// TIA Portal project "2Nastri1Ruota" (V17)
// Vorlageprojekt für das Buch mit Zielsystem S7-1200

(* hardware
DEVICE "S7-1200-Station_1"  S7-1200 Station
   slot 0: "Baugruppenträger_0"  Rack  V1.0
   slot 1: "PLC_1"  CPU 1211C DC/DC/DC  6ES7 211-1AE40-0XB0  V4.1
*)

// ===== PLC "PLC_1"  CPU 1211C DC/DC/DC =====

VAR_GLOBAL   // PLC tag table "Standard-Variablentabelle"
   "S11" AT %I0.0 : Bool;
   "S12" AT %I0.1 : Bool;
   "S21" AT %I0.2 : Bool;
   "S22" AT %I0.3 : Bool;
   "AVA1" AT %Q0.0 : Bool;
   "AVA2" AT %Q0.1 : Bool;
   "AVAN" AT %Q0.2 : Bool;
   "Lim_R1" AT %I0.4 : Bool;
   "Lim_R2" AT %I0.5 : Bool;
   "SIN" AT %I0.6 : Bool;
   "SFN" AT %I0.7 : Bool;
   "RUO" AT %Q0.3 : Bool;
END_VAR

DATA_BLOCK "Sistema_DB"   // DB1
{ S7_Optimized_Access := 'TRUE' }
VERSION : 0.1
// stored: InstanceOfName Sistema
"Sistema"
BEGIN
END_DATA_BLOCK

FUNCTION_BLOCK "Nastro"   // FB1, LAD
{ S7_Optimized_Access := 'TRUE' }
VERSION : 0.1
   VAR_INPUT
      SI : Bool;
      SF : Bool;
      P_DOPO : Bool;
   END_VAR
   VAR_OUTPUT
      AVA : Bool;
      P_CONS : Bool;
      P_ACC : Bool;
      CONS_OK : Bool;
   END_VAR
   VAR
      F0 : Bool;
      F1 : Bool;
      TR0 : Bool;
      TR1 : Bool;
      INIT : Bool;
   END_VAR
   VAR_TEMP   // added for the SCL form of the ladder/FBD networks
      _w1 : Bool;
   END_VAR
BEGIN

REGION Network 1: INIZIALIZZAZIONE
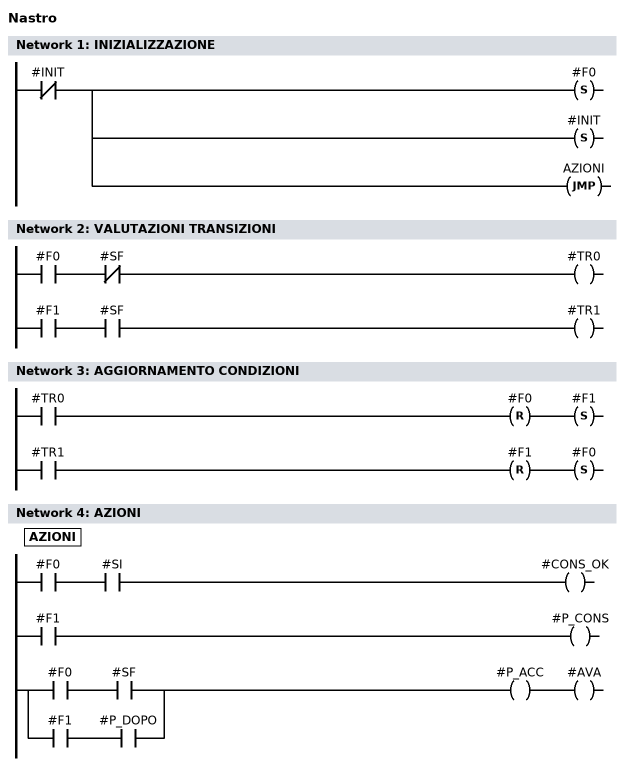
   RUNG wire#powerrail
      I_Contact( #INIT )
      wire#w1
      S_Coil( #F0 )
   END_RUNG
   RUNG wire#w1
      S_Coil( #INIT )
   END_RUNG
   RUNG wire#w1
      JumpCoil( AZIONI )
   END_RUNG
   // the same network as SCL:
   IF NOT #INIT THEN #F0 := TRUE; END_IF;
   #_w1 := NOT #INIT;
   IF #_w1 THEN
       #INIT := TRUE;
       GOTO AZIONI;
   END_IF;
END_REGION

REGION Network 2: VALUTAZIONI TRANSIZIONI
   RUNG wire#powerrail
      Contact( #F0 )
      I_Contact( #SF )
      Coil( #TR0 )
   END_RUNG
   RUNG wire#powerrail
      Contact( #F1 )
      Contact( #SF )
      Coil( #TR1 )
   END_RUNG
   // the same network as SCL:
   #TR0 := #F0 AND NOT #SF;
   #TR1 := #F1 AND #SF;
END_REGION

REGION Network 3: AGGIORNAMENTO CONDIZIONI
   RUNG wire#powerrail
      Contact( #TR0 )
      R_Coil( #F0 )
      S_Coil( #F1 )
   END_RUNG
   RUNG wire#powerrail
      Contact( #TR1 )
      R_Coil( #F1 )
      S_Coil( #F0 )
   END_RUNG
   // the same network as SCL:
   IF #TR0 THEN
       #F0 := FALSE;
       #F1 := TRUE;
   END_IF;
   IF #TR1 THEN
       #F1 := FALSE;
       #F0 := TRUE;
   END_IF;
END_REGION

REGION Network 4: AZIONI
   Label( AZIONI )
   RUNG wire#powerrail
      Contact( #F0 )
      Contact( #SI )
      Coil( #CONS_OK )
   END_RUNG
   RUNG wire#powerrail
      Contact( #F1 )
      Coil( #P_CONS )
   END_RUNG
   RUNG wire#powerrail
      Contact( #F0 )
      Contact( #SF )
      wire#w1
      Coil( #P_ACC )
      Coil( #AVA )
   END_RUNG
   RUNG wire#powerrail
      Contact( #F1 )
      Contact( #P_DOPO )
   END_RUNG wire#w1
   // the same network as SCL:
   AZIONI:
   #CONS_OK := #F0 AND #SI;
   #P_CONS := #F1;
   #P_ACC := (#F0 AND #SF) OR (#F1 AND #P_DOPO);
   #AVA := #P_ACC;
END_REGION
END_FUNCTION_BLOCK

FUNCTION_BLOCK "Ruota"   // FB2, LAD
{ S7_Optimized_Access := 'TRUE' }
VERSION : 0.1
   VAR_INPUT
      Lim_R1 : Bool;
      Lim_R2 : Bool;
      SI : Bool;
      SF : Bool;
      P_PRIMA : Bool;
      P_DOPO : Bool;
      CONS_OK : Bool;
   END_VAR
   VAR_OUTPUT
      RUOTA : Bool;
      IND : Bool;
      AVA : Bool;
      P_ACC : Bool;
      P_CONS : Bool;
   END_VAR
   VAR
      INIT : Bool;
      F0 : Bool;
      F1 : Bool;
      F2 : Bool;
      F3 : Bool;
      TR0 : Bool;
      TR1 : Bool;
      TR2 : Bool;
      TR3 : Bool;
      "MEMO-1" : Bool;
      "MEMO-2" : Bool;
   END_VAR
   VAR_TEMP   // added for the SCL form of the ladder/FBD networks
      _w1 : Bool;
      _w2 : Bool;
   END_VAR
BEGIN

REGION Network 1: INIZIALIZZAZIONE
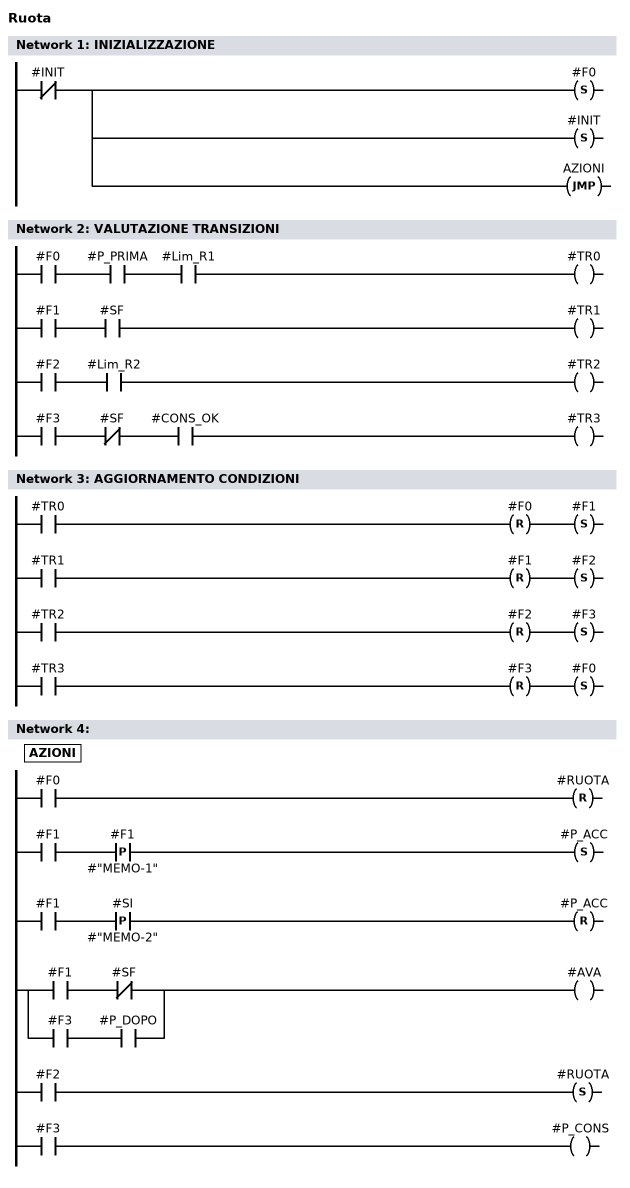
   RUNG wire#powerrail
      I_Contact( #INIT )
      wire#w1
      S_Coil( #F0 )
   END_RUNG
   RUNG wire#w1
      S_Coil( #INIT )
   END_RUNG
   RUNG wire#w1
      JumpCoil( AZIONI )
   END_RUNG
   // the same network as SCL:
   IF NOT #INIT THEN #F0 := TRUE; END_IF;
   #_w1 := NOT #INIT;
   IF #_w1 THEN
       #INIT := TRUE;
       GOTO AZIONI;
   END_IF;
END_REGION

REGION Network 2: VALUTAZIONE TRANSIZIONI
   RUNG wire#powerrail
      Contact( #F0 )
      Contact( #P_PRIMA )
      Contact( #Lim_R1 )
      Coil( #TR0 )
   END_RUNG
   RUNG wire#powerrail
      Contact( #F1 )
      Contact( #SF )
      Coil( #TR1 )
   END_RUNG
   RUNG wire#powerrail
      Contact( #F2 )
      Contact( #Lim_R2 )
      Coil( #TR2 )
   END_RUNG
   RUNG wire#powerrail
      Contact( #F3 )
      I_Contact( #SF )
      Contact( #CONS_OK )
      Coil( #TR3 )
   END_RUNG
   // the same network as SCL:
   #TR0 := #F0 AND #P_PRIMA AND #Lim_R1;
   #TR1 := #F1 AND #SF;
   #TR2 := #F2 AND #Lim_R2;
   #TR3 := #F3 AND NOT #SF AND #CONS_OK;
END_REGION

REGION Network 3: AGGIORNAMENTO CONDIZIONI
   RUNG wire#powerrail
      Contact( #TR0 )
      R_Coil( #F0 )
      S_Coil( #F1 )
   END_RUNG
   RUNG wire#powerrail
      Contact( #TR1 )
      R_Coil( #F1 )
      S_Coil( #F2 )
   END_RUNG
   RUNG wire#powerrail
      Contact( #TR2 )
      R_Coil( #F2 )
      S_Coil( #F3 )
   END_RUNG
   RUNG wire#powerrail
      Contact( #TR3 )
      R_Coil( #F3 )
      S_Coil( #F0 )
   END_RUNG
   // the same network as SCL:
   IF #TR0 THEN
       #F0 := FALSE;
       #F1 := TRUE;
   END_IF;
   IF #TR1 THEN
       #F1 := FALSE;
       #F2 := TRUE;
   END_IF;
   IF #TR2 THEN
       #F2 := FALSE;
       #F3 := TRUE;
   END_IF;
   IF #TR3 THEN
       #F3 := FALSE;
       #F0 := TRUE;
   END_IF;
END_REGION

REGION Network 4
   Label( AZIONI )
   RUNG wire#powerrail
      Contact( #F0 )
      R_Coil( #RUOTA )
   END_RUNG
   RUNG wire#powerrail
      Contact( #F1 )
      P_Contact(operand := #F1, bit := #"MEMO-1")
      S_Coil( #P_ACC )
   END_RUNG
   RUNG wire#powerrail
      Contact( #F1 )
      P_Contact(operand := #SI, bit := #"MEMO-2")
      R_Coil( #P_ACC )
   END_RUNG
   RUNG wire#powerrail
      Contact( #F1 )
      I_Contact( #SF )
      wire#w1
      Coil( #AVA )
   END_RUNG
   RUNG wire#powerrail
      Contact( #F3 )
      Contact( #P_DOPO )
   END_RUNG wire#w1
   RUNG wire#powerrail
      Contact( #F2 )
      S_Coil( #RUOTA )
   END_RUNG
   RUNG wire#powerrail
      Contact( #F3 )
      Coil( #P_CONS )
   END_RUNG
   // the same network as SCL:
   AZIONI:
   IF #F0 THEN #RUOTA := FALSE; END_IF;
   #_w1 := #F1 AND #F1 AND NOT #"MEMO-1";   // rising edge of #F1
   #"MEMO-1" := #F1;
   IF #_w1 THEN #P_ACC := TRUE; END_IF;
   #_w2 := #F1 AND #SI AND NOT #"MEMO-2";   // rising edge of #SI
   #"MEMO-2" := #SI;
   IF #_w2 THEN #P_ACC := FALSE; END_IF;
   #AVA := (#F1 AND NOT #SF) OR (#F3 AND #P_DOPO);
   IF #F2 THEN #RUOTA := TRUE; END_IF;
   #P_CONS := #F3;
END_REGION
END_FUNCTION_BLOCK

FUNCTION_BLOCK "Sistema"   // FB3, FBD
{ S7_Optimized_Access := 'TRUE' }
VERSION : 0.1
   VAR
      Nastro1 : "Nastro";
      Nastro2 : "Nastro";
      Ruota : "Ruota";
   END_VAR
BEGIN

REGION Network 1
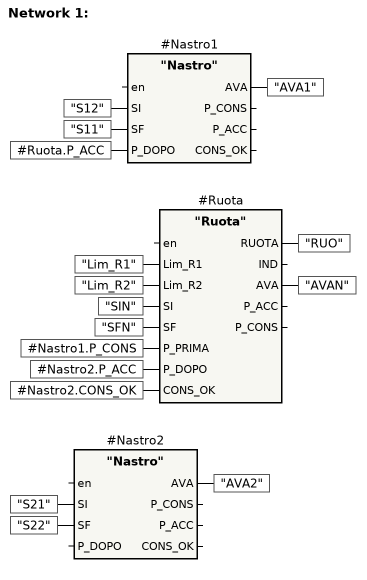
   #Nastro1(SI := "S12", SF := "S11", P_DOPO := #Ruota.P_ACC, AVA => "AVA1");   // "Nastro"
   #Ruota(Lim_R1 := "Lim_R1",   // "Ruota"
          Lim_R2 := "Lim_R2",
          SI := "SIN",
          SF := "SFN",
          P_PRIMA := #Nastro1.P_CONS,
          P_DOPO := #Nastro2.P_ACC,
          CONS_OK := #Nastro2.CONS_OK,
          RUOTA => "RUO",
          AVA => "AVAN");
   #Nastro2(SI := "S21", SF := "S22", AVA => "AVA2");   // "Nastro"
END_REGION
END_FUNCTION_BLOCK

FUNCTION "MHJ-PLC-Lab-Function-S71200" : Void   // FC9000, SCL
{ S7_Optimized_Access := 'TRUE' }
VERSION : 0.1
   VAR_TEMP
      rdTimeReturn : Int;
      outputTime : DTL;
      SyncVal : Byte;
      forVal : Int;
      forVal_2 : Int;
      Value : Byte;
   END_VAR
   VAR CONSTANT
      CompVal : Byte := 16#34;
      Value_01 : Byte := 16#11;
      Value_01_DW : DWord := 16#A165_D992;
      Value_02_DW : DWord := 16#58BE_4401;
   END_VAR
BEGIN

   #Value:=PEEK(area := 16#82,
        dbNumber := 0,
        byteOffset := 511);
   #Value := #Value + 1;

   POKE(area := 16#82,
        dbNumber := 0,
        byteOffset := 511,
        value := #Value);

   POKE(area:=16#81,
        dbNumber:=0,
        byteOffset:=1016,
        value:=#Value_01_DW);
   POKE(area := 16#81,
        dbNumber := 0,
        byteOffset := 1020,
        value := #Value_02_DW);

   POKE(area := 16#81,
        dbNumber := 0,
        byteOffset := 511,
        value := B#16#00);

   FOR #forVal := 0 TO 120 DO
       FOR #forVal_2:=0 TO 10 DO
           #rdTimeReturn:=RD_SYS_T(#outputTime);
           #rdTimeReturn := WR_SYS_T(#outputTime);
           #rdTimeReturn := RD_SYS_T(#outputTime);
           #rdTimeReturn := WR_SYS_T(#outputTime);
       END_FOR;
       #SyncVal:= PEEK(area := 16#81,
                      dbNumber := 0,
                      byteOffset := 511);
       IF #SyncVal = #CompVal THEN
          GOTO M_1;
       END_IF;
   END_FOR;
   RETURN;

   M_1:
   POKE(area := 16#81,
        dbNumber := 0,
        byteOffset := 511,
        value := B#16#0);
END_FUNCTION

ORGANIZATION_BLOCK "Main"   // OB1, FBD, ProgramCycle
TITLE = "Main Program Sweep (Cycle)"
{ S7_Optimized_Access := 'TRUE' }
VERSION : 0.1
   VAR_INPUT
      Initial_Call : Bool;   // Initial call of this OB
      Remanence : Bool;   // =True, if remanent data are available
   END_VAR
BEGIN

REGION Network 1: Konnektierungsbaustein für PLC-Lab
   // Im Netzwerk 1 wird der Konnektierungsbaustein für PLC-Lab aufgerufen.
   // Dieser Aufruf darf nicht entfernt werden!
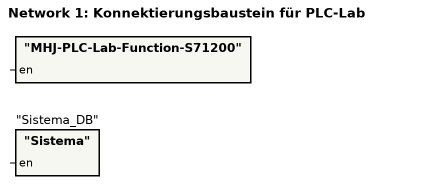
   "MHJ-PLC-Lab-Function-S71200"();
   "Sistema_DB"();   // "Sistema"
END_REGION

REGION Network 2: Ihr Programm
   // Schreiben Sie ab Netzwerk 2 Ihr Programm
END_REGION
END_ORGANIZATION_BLOCK